(* IEC 61131-3 sources: AXOpen/src/components.festo.drives/ctrl/src/PROFIdrive, 6 files *)

(* ---- AxoPROFIdriveParametrization.st ---- *)
USING AXOpen.Core;
USING Siemens.Simatic.DistributedIO;

NAMESPACE AXOpen.Components.Festo.Drives
    {S7.extern=ReadWrite}
    CLASS AxoPROFIdriveParametrization
        VAR PUBLIC
            {#ix-attr:[Container(Layout.Wrap)]}
            {#ix-attr:[Group(GroupLayout.GroupBox)]}
            {#ix-set:AttributeName = "<#Inputs#>"}
            Inputs				:	AxoPROFIdriveParametrizationIn;
            {#ix-attr:[Container(Layout.Wrap)]}
            {#ix-attr:[Group(GroupLayout.GroupBox)]}
            {#ix-set:AttributeName = "<#Outputs#>"}
            {#ix-attr:[ReadOnly()]}
            Outputs				:	AxoPROFIdriveParametrizationOut;
        END_VAR
    END_CLASS
END_NAMESPACE

(* ---- AxoPROFIdriveParametrizationIn.st ---- *)
USING AXOpen.Core;
USING Siemens.Simatic.DistributedIO;

NAMESPACE AXOpen.Components.Festo.Drives
    {S7.extern=ReadWrite}
    CLASS AxoPROFIdriveParametrizationIn
        VAR PUBLIC
            {#ix-attr:[Container(Layout.Stack)]}
            {#ix-set:AttributeName = "<#Enable#>"}
            Enable          :   BOOL;
            {#ix-set:AttributeName = "<#ReadWrite#>"}
            ReadWrite       :   BOOL;
            {#ix-set:AttributeName = "<#ParameterNo#>"}
            ParameterNo     :   INT;
            {#ix-set:AttributeName = "<#Subindex#>"}
            Subindex        :   INT;
            {#ix-set:AttributeName = "<#AxisNo#>"}
            AxisNo	        :   BYTE := BYTE#1;
            {#ix-set:AttributeName = "<#HardwareId#>"}
            HardwareId	    :   UINT;
            {#ix-set:AttributeName = "<#ValueWriteREAL#>"}
            ValueWriteREAL  :   REAL;
            {#ix-set:AttributeName = "<#ValueWriteLINT#>"}
            ValueWriteLINT  :   LINT;
            {#ix-set:AttributeName = "<#ValueWriteBOOL#>"}
            ValueWriteBOOL  :   BOOL;
        END_VAR
    END_CLASS
END_NAMESPACE

(* ---- AxoPROFIdriveParametrizationOut.st ---- *)
USING AXOpen.Core;
USING Siemens.Simatic.DistributedIO;

NAMESPACE AXOpen.Components.Festo.Drives
    {S7.extern=ReadWrite}
    CLASS AxoPROFIdriveParametrizationOut
        VAR PUBLIC
            {#ix-attr:[Container(Layout.Stack)]}
            {#ix-set:AttributeName = "<#ValueReadREAL#>"}
            ValueReadREAL  :   REAL;
            {#ix-set:AttributeName = "<#ValueReadLINT#>"}
            ValueReadLINT  :   LINT;
            {#ix-set:AttributeName = "<#ValueReadBOOL#>"}
            ValueReadBOOL  :   BOOL;
            {#ix-set:AttributeName = "<#Busy#>"}
            Busy	:   BOOL;
            {#ix-set:AttributeName = "<#Done#>"}
            Done	:   BOOL;
            {#ix-set:AttributeName = "<#Error#>"}
            Error	:   BOOL;
            {#ix-set:AttributeName = "<#ErrorId#>"}
            ErrorId :	DWORD;
        END_VAR

    END_CLASS
END_NAMESPACE

(* ---- AxoReadWritePROFIdriveParameter.st ---- *)
USING AXOpen.Core;
USING Siemens.Simatic.S71500.DistributedIO;

NAMESPACE AXOpen.Components.Festo.Drives
    {S7.extern=ReadWrite}
    CLASS AxoReadWritePROFIdriveParameter EXTENDS AXOpen.Core.AxoObject
        VAR PUBLIC
            {#ix-attr:[Container(Layout.Wrap)]}
            {#ix-attr:[Group(GroupLayout.GroupBox)]}
            {#ix-set:AttributeName = "<#Inputs#>"}
            Inputs				:	AxoPROFIdriveParametrizationIn;
            {#ix-attr:[Container(Layout.Wrap)]}
            {#ix-attr:[Group(GroupLayout.GroupBox)]}
            {#ix-set:AttributeName = "<#Outputs#>"}
            {#ix-attr:[ReadOnly()]}
            Outputs				:	AxoPROFIdriveParametrizationOut;
        END_VAR

        VAR PRIVATE
            Enable_PV   :   BOOL;

            Busy_	:   BOOL;
            Done_	:   BOOL;
            Error_	:   BOOL;
            ErrorId_:	DWORD;
            StartTimer : BOOL;
            StartRW : BOOL;

            AxoOnDelatTimer :  AXOpen.Timers.OnDelayTimer;

            RW_Data         :   ARRAY[0..9] OF BYTE;
            WR_Data         :   ARRAY[0..19] OF BYTE;
            RD_Data         :   ARRAY[0..13] OF BYTE;
            RW_Status        :	DWORD;
            WR_Status        :	DWORD;
            RD_Status        :	DWORD;

            ReadRecord_     :   ReadRecord;
            WriteRecord_    :   WriteRecord;
            ErrorCounter    :	UINT;

            LengthRead      :	UINT;
            State           :   INT;
            ReqRef          :   BYTE;
            wordhlp         :   WORD;

            _lenght     :   UINT;
            tmpWord     :   WORD;
            tmpSINT     :   SINT;
            tmpINT      :   INT;
            tmpDINT     :   DINT;
            tmpDWORD    :   DWORD;
            tmpLINT     :   LINT;
        END_VAR

        VAR CONSTANT PRIVATE
            LenHeader	    :   UINT    :=	UINT#4;
            LenRequest	    :   UINT    :=  UINT#6;
            LenWrite	    :   UINT    :=  UINT#16;
            LenRead	        :   UINT    :=  UINT#10;
            PD_Error	    :   DWORD	:=  DWORD#16#4000_0000;
            MaxRetryCounter	:   UINT    :=	UINT#150;

        END_VAR

        METHOD PUBLIC OVERRIDE Run
            VAR_INPUT
                inParent : IAxoObject;
            END_VAR
            VAR
                i : INT;
            END_VAR

            SUPER.Run(inParent);

            //**********************************************
            // THIS.Execute();
            //*****************Execute inline***************
                //Check the Inputs
                IF Inputs.HardwareId = WORD#0 THEN
                    Error_ := TRUE;
                    ErrorId_ := DWORD#16#00001010;    //Inputs.HardwareId = 0
                    RETURN;
                END_IF;

                //Timer
                AxoOnDelatTimer.OnDelay(THIS, StartTimer,T#100MS);

                IF AxoOnDelatTimer.output THEN
                    StartRW := TRUE;
                    StartTimer := FALSE;
                END_IF;

                IF State = 0 THEN //Wait for start trigger
                    IF Inputs.Enable AND NOT Enable_PV THEN
                        StartRW := TRUE;
                        State := 10;
                        Outputs.Busy := TRUE;
                    END_IF;
                END_IF;

                IF State = 10 THEN
                    (* ------------------ HEADER --------------------*)
                    //Request reference starts with 1 and will count up
                    RW_Data[0] := ReqRef;
                    // Requst ID = 1 (Request Parameter)
                    RW_Data[1] := BYTE#1;
                    //Fill the Axis number
                    RW_Data[2] := Inputs.AxisNo;
                    // Single parameter access
                    RW_Data[3] := BYTE#1;
                    (* ------------------ Parameter address ------------*)
                    //Attribute
                    RW_Data[4]:= BYTE#16#10;
                    //ElemNo.
                    RW_Data[5] := BYTE#1;
                    // Assign PNU
                    RW_Data[6] := Inputs.ParameterNo.%B1;
                    RW_Data[7] := Inputs.ParameterNo.%B0;
                    // Assign Subindex
                    RW_Data[8] := Inputs.Subindex.%B1;
                    RW_Data[9] := Inputs.Subindex.%B0;

                    // Lenght of the telegramm to be send
                    _lenght := LenHeader + LenRequest;

                    WriteRecord_(request    :=  StartRW,
                                id          :=  Inputs.HardwareId,
                                index       :=  16#b02e,
                                length      :=  _lenght,
                                record      :=  RW_Data,
                                status      =>  WR_Status);

                    IF WriteRecord_.DONE THEN
                        ErrorCounter := UINT#0;
                        //delete old response values
                        FOR i := 0 TO 13 DO
                            RD_Data[i] := BYTE#0;
                        END_FOR;

                        IF NOT Inputs.ReadWrite THEN
                            //Read parameter
                            State := 20;
                        ELSE
                            //Write parameter
                            State := 50;
                        END_IF;
                    ELSIF WriteRecord_.ERROR THEN
                        tmpWord := TO_WORD(TO_DINT(WR_Status)/256);
                        wordhlp := tmpWord;
                        //try it again
                        IF ((tmpWord = WORD#16#80A7) OR (tmpWord = WORD#16#80B5) OR (tmpWord = WORD#16#80C0) OR (tmpWord = WORD#16#80C1) OR (tmpWord = WORD#16#80C2)
                            OR (tmpWord = WORD#16#80C3) OR (tmpWord = WORD#16#80C4)) AND (ErrorCounter < MaxRetryCounter) THEN
                            ErrorCounter := ErrorCounter + UINT#1;
                            StartRW := FALSE;
                            StartTimer := TRUE;
                        ELSE
                            State := 70;
                        END_IF;

                    END_IF;
                END_IF;

                IF State = 20 THEN  //Read Parameter
                    // Lenght of the telegramm for reading
                    _lenght := LenHeader + LenRead;

                    ReadRecord_(request     :=  StartRW,
                                id          :=  Inputs.HardwareId,
                                index       :=  16#b02e,
                                maxLength   :=  _lenght,
                                record      :=  RD_Data,
                                status      =>  RD_Status,
                                length      =>  LengthRead);

                    IF ReadRecord_.VALID AND NOT ReadRecord_.BUSY THEN
                        ErrorCounter := UINT#0;
                        State := 30;
                    ELSIF ReadRecord_.ERROR THEN
                        tmpWord := TO_WORD(TO_DINT(RD_Status) / 256);
                        wordhlp := tmpWord;
                        //try it again
                        IF ((tmpWord = WORD#16#80A7) OR (tmpWord = WORD#16#80B5) OR (tmpWord = WORD#16#80C0) OR (tmpWord = WORD#16#80C1) OR (tmpWord = WORD#16#80C2)
                            OR (tmpWord = WORD#16#80C3) OR (tmpWord = WORD#16#80C4)) AND (ErrorCounter < MaxRetryCounter) THEN
                            ErrorCounter := ErrorCounter + UINT#1;
                            StartRW := FALSE;
                            StartTimer := TRUE;
                        ELSE
                            State := 80;
                        END_IF;
                    END_IF;
                END_IF;

                IF State = 30 THEN //Reading finished successfull

                    CASE TO_INT(RD_Data[4]) OF //Format
                        0:  //reserved
                            Outputs.ValueReadREAL := REAL#0.0;
                            Outputs.ValueReadLINT := LINT#0;
                            Outputs.ValueReadBOOL := FALSE;

                            Outputs.ErrorId := DWORD#16#1001;    //reserved DataType
                            // #Error
                            State := 200;

                        1:  // BOOLEAN
                            //copy the value to the output
                            Outputs.ValueReadREAL := 0;
                            Outputs.ValueReadLINT := 0;
                            Outputs.ValueReadBOOL := TO_BOOL(RD_Data[6]);

                            // no error
                            State := 100;

                        2:  //SINT8
                            tmpSINT := TO_SINT(RD_Data[6]);
                            //copy the value to the output
                            Outputs.ValueReadREAL := 0;
                            Outputs.ValueReadLINT := (TO_LINT(tmpSINT));
                            Outputs.ValueReadBOOL := FALSE;

                            // no error
                            State := 100;

                        3:  //SINT16
                            tmpINT.%B0 := RD_Data[7];
                            tmpINT.%B1 := RD_Data[6];

                            //copy the value to the output
                            Outputs.ValueReadREAL := 0;
                            Outputs.ValueReadLINT := TO_LINT(tmpINT);
                            Outputs.ValueReadBOOL := FALSE;

                            // no #Error
                            State := 100;

                        4:  //SINT32
                            tmpDINT.%B0 := RD_Data[9];
                            tmpDINT.%B1 := RD_Data[8];
                            tmpDINT.%B2 := RD_Data[7];
                            tmpDINT.%B3 := RD_Data[6];

                            //copy the value to the output
                            Outputs.ValueReadREAL := 0;
                            Outputs.ValueReadLINT := TO_LINT(tmpDINT);
                            Outputs.ValueReadBOOL := FALSE;

                            // no #Error
                            State := 100;

                        5, 65: //USINT8(5) or BYTE(65)
                            //copy the value to the output
                            Outputs.ValueReadREAL := 0;
                            Outputs.ValueReadLINT := (TO_LINT(RD_Data[6]));
                            Outputs.ValueReadBOOL := FALSE;

                            // no error
                            State := 100;

                        6, 66: //UINT16(6) or WORD(66)
                            tmpWord.%B0 := RD_Data[7];
                            tmpWord.%B1 := RD_Data[6];

                            //copy the value to the output
                            Outputs.ValueReadREAL := 0;
                            Outputs.ValueReadLINT := TO_LINT(tmpWord);
                            Outputs.ValueReadBOOL := FALSE;

                            // no #Error
                            State := 100;

                        7, 67: //UDINT32(7) or DWORD(67)
                            tmpDWord.%B0 := RD_Data[9];
                            tmpDWord.%B1 := RD_Data[8];
                            tmpDWord.%B2 := RD_Data[7];
                            tmpDWord.%B3 := RD_Data[6];

                            //copy the value to the output
                            Outputs.ValueReadREAL := 0;
                            Outputs.ValueReadLINT := TO_LINT(tmpDWord);
                            Outputs.ValueReadBOOL := FALSE;

                            // no #Error
                            State := 100;

                        8:  //FLOAT32
                            tmpDWord.%B0 := RD_Data[9];
                            tmpDWord.%B1 := RD_Data[8];
                            tmpDWord.%B2 := RD_Data[7];
                            tmpDWord.%B3 := RD_Data[6];

                            //copy the value to the output
                            Outputs.ValueReadREAL := TO_REAL(tmpDWord);
                            Outputs.ValueReadLINT := 0;
                            Outputs.ValueReadBOOL := FALSE;

                            // no #Error
                            State := 100;

                        10:  //OctetString
                            tmpINT.%B0 := RD_Data[6];
                            tmpINT.%B1 := RD_Data[7];

                            //copy the value to the output
                            Outputs.ValueReadREAL := 0;
                            Outputs.ValueReadLINT := TO_LINT(tmpINT);
                            Outputs.ValueReadBOOL := FALSE;

                            // no #Error
                            State := 100;

                        55, 56:  //LINT, ULINT
                            tmpLINT.%B0 :=RD_Data[13];
                            tmpLINT.%B1 :=RD_Data[12];
                            tmpLINT.%B2 :=RD_Data[11];
                            tmpLINT.%B3 :=RD_Data[10];
                            tmpLINT.%B4 :=RD_Data[9];
                            tmpLINT.%B5 :=RD_Data[8];
                            tmpLINT.%B6 :=RD_Data[7];
                            tmpLINT.%B7 :=RD_Data[6];

                            //copy the value to the output
                            Outputs.ValueReadREAL := 0;
                            Outputs.ValueReadLINT := tmpLINT;
                            Outputs.ValueReadBOOL := FALSE;

                            // no #Error
                            State := 100;

                        68:  //Error
                            tmpDWord.%B0 := RD_Data[7];
                            tmpDWord.%B1 := RD_Data[6];
                            Outputs.ErrorId := tmpDWord OR PD_Error;

                            //copy the value to the output
                            Outputs.ValueReadREAL := 0;
                            Outputs.ValueReadLINT := 0;
                            Outputs.ValueReadBOOL := FALSE;

                            // #Error
                            State := 200;

                        ELSE
                            Outputs.ValueReadREAL := 0;
                            Outputs.ValueReadLINT := 0;
                            Outputs.ValueReadBOOL := FALSE;

                            Outputs.ErrorId := DWORD#16#1000;    //unknown DataType
                            // #Error
                            State := 200;
                    END_CASE;
                END_IF;

                IF State = 50 THEN //Write Parameter (First Read dataset then write dataset)
                    // Lenght of the telegramm for reading
                    _lenght := LenHeader + LenRead;

                    ReadRecord_(request     :=  StartRW,
                                id          :=  Inputs.HardwareId,
                                index       :=  16#b02e,
                                maxLength   :=  _lenght,
                                record      :=  RD_Data,
                                status      =>  RD_Status,
                                length      =>  LengthRead);

                    IF ReadRecord_.VALID AND NOT ReadRecord_.BUSY THEN
                        ErrorCounter := UINT#0;
                        State := 55;
                    ELSIF ReadRecord_.ERROR THEN
                        tmpWord := TO_WORD(TO_DINT(RD_Status)/256);
                        wordhlp := tmpWord;
                        //try it again
                        IF ((tmpWord = WORD#16#80A7) OR (tmpWord = WORD#16#80B5) OR (tmpWord = WORD#16#80C0) OR (tmpWord = WORD#16#80C1) OR (tmpWord = WORD#16#80C2)
                            OR (tmpWord = WORD#16#80C3) OR (tmpWord = WORD#16#80C4)) AND (ErrorCounter < MaxRetryCounter) THEN
                            ErrorCounter := ErrorCounter + UINT#1;
                            StartRW := false;
                            StartTimer := TRUE;
                        ELSE
                            State := 80;
                        END_IF;
                    END_IF;
                END_IF;

                IF State = 55 THEN //Reading finished
                    CASE TO_INT(RD_Data[4]) OF // Format
                        0:  //reserved
                            Outputs.ValueReadREAL := 0;
                            Outputs.ValueReadLINT := 0;
                            Outputs.ValueReadBOOL := FALSE;

                            Outputs.ErrorId := DWORD#16#1001;    //reserved DataType
                            // #Error
                            State := 200;

                        1, 2, 3, 4, 5, 6, 7, 8, 55, 56, 65, 66, 67:
                            State := 60;

                        68:  //Error
                            tmpDWord.%B0 := RD_Data[7];
                            tmpDWord.%B1 := RD_Data[6];
                            Outputs.ErrorId := tmpDWord OR PD_Error;

                            //copy the value to the output
                            Outputs.ValueReadREAL := 0;
                            Outputs.ValueReadLINT := 0;
                            Outputs.ValueReadBOOL := FALSE;

                            // #Error
                            State := 200;

                        ELSE
                            Outputs.ValueReadREAL := 0;
                            Outputs.ValueReadLINT := 0;
                            Outputs.ValueReadBOOL := FALSE;

                            Outputs.ErrorId := DWORD#16#1000;    //unknown DataType
                            // #Error
                            State := 200;
                    END_CASE;
                END_IF;

                IF State = 60 THEN //reading Done from Write request
                    (* ------------------ HEADER --------------------*)
                    //Request reference starts with 1 and will count up
                    WR_Data[0] := TO_BYTE(TO_INT(ReqRef) + 1);
                    // Requst ID = 2 (Change Parameter)
                    WR_Data[1] := BYTE#2;
                    //Fill the Axis number
                    WR_Data[2] := Inputs.AxisNo;
                    // Single parameter access
                    WR_Data[3] := BYTE#1;
                    (* ------------------ DATA --------------------*)
                    // Attribute
                    WR_Data[4] := BYTE#16#10;
                    // Single Access
                    WR_Data[5] := BYTE#1;
                    // PNU
                    WR_Data[6] := Inputs.ParameterNo.%B1;
                    WR_Data[7] := Inputs.ParameterNo.%B0;
                    // Subindex
                    WR_Data[8] := Inputs.Subindex.%B1;
                    WR_Data[9] := Inputs.Subindex.%B0;
                    //Format
                    WR_Data[10] := RD_Data[4];
                    //No. Values
                    WR_Data[11] := BYTE#1;
                    //erase send buffer
                    FOR i := 12 TO 19 DO
                        WR_Data[i] := BYTE#0;
                    END_FOR;

                    CASE TO_INT(RD_Data[4]) OF //Format
                        0:  //reserved
                            Outputs.ValueReadREAL := 0;
                            Outputs.ValueReadLINT := 0;
                            Outputs.ValueReadBOOL := FALSE;

                            Outputs.ErrorId := DWORD#16#1001;    //reserved DataType
                            // #Error
                            State := 200;

                        1:  //BOOL
                            WR_Data[12] := TO_BYTE(Inputs.ValueWriteBOOL);

                        2, 5, 65:  //SINT8, USINT8, BYTE
                            WR_Data[12] := TO_BYTE(Inputs.ValueWriteLINT);

                        3, 6, 66:  //SINT16, UINT16, WORD
                            WR_Data[12] := Inputs.ValueWriteLINT.%B1;
                            WR_Data[13] := Inputs.ValueWriteLINT.%B0;

                        4, 7, 67: //SINT32, UDINT32, DWORD
                            WR_Data[12] := Inputs.ValueWriteLINT.%B3;
                            WR_Data[13] := Inputs.ValueWriteLINT.%B2;
                            WR_Data[14] := Inputs.ValueWriteLINT.%B1;
                            WR_Data[15] := Inputs.ValueWriteLINT.%B0;

                        8:  //FLOAT32
                            tmpDWORD    :=  TO_DWORD(Inputs.ValueWriteREAL);
                            WR_Data[12] := tmpDWORD.%B3;
                            WR_Data[13] := tmpDWORD.%B2;
                            WR_Data[14] := tmpDWORD.%B1;
                            WR_Data[15] := tmpDWORD.%B0;

                        55, 56:  //SINT64
                            WR_Data[12] := Inputs.ValueWriteLINT.%B7;
                            WR_Data[13] := Inputs.ValueWriteLINT.%B6;
                            WR_Data[14] := Inputs.ValueWriteLINT.%B5;
                            WR_Data[15] := Inputs.ValueWriteLINT.%B4;
                            WR_Data[16] := Inputs.ValueWriteLINT.%B3;
                            WR_Data[17] := Inputs.ValueWriteLINT.%B2;
                            WR_Data[18] := Inputs.ValueWriteLINT.%B1;
                            WR_Data[19] := Inputs.ValueWriteLINT.%B0;

                    END_CASE;

                    //goto the next step
                    State := 61;
                END_IF;

                IF State = 61 THEN //send the write Request
                    // Lenght of the telegramm to be send
                    _lenght := LenHeader + LenWrite;

                    WriteRecord_(request    :=  StartRW,
                                id          :=  Inputs.HardwareId,
                                index       :=  16#b02e,
                                length      :=  _lenght,
                                record      :=  WR_Data,
                                status      =>  RW_Status);

                    IF WriteRecord_.DONE THEN
                        State := 62;
                    ELSIF WriteRecord_.ERROR THEN
                        tmpWord := TO_WORD(TO_DINT(RW_Status)/256);
                        wordhlp := tmpWord;
                        //try it again
                        IF ((tmpWord = WORD#16#80A7) OR (tmpWord = WORD#16#80B5) OR (tmpWord = WORD#16#80C0) OR (tmpWord = WORD#16#80C1) OR (tmpWord = WORD#16#80C2)
                            OR (tmpWord = WORD#16#80C3) OR (tmpWord = WORD#16#80C4)) AND (ErrorCounter < MaxRetryCounter) THEN
                            ErrorCounter := ErrorCounter + UINT#1;
                            StartRW := FALSE;
                            StartTimer := TRUE;
                        ELSE
                            State := 90;
                        END_IF;
                    END_IF;
                END_IF;

                IF State = 62 THEN //Read the answer of the write request

                    //delete old response values
                    FOR i := 0 TO 13 DO
                        RD_Data[i] := BYTE#0;
                    END_FOR;

                    // Lenght of the telegramm for reading
                    _lenght := LenHeader + LenRead;

                    ReadRecord_(request     :=  StartRW,
                                id          :=  Inputs.HardwareId,
                                index       :=  16#b02e,
                                maxLength   :=  _lenght,
                                record      :=  RD_Data,
                                status      =>  RD_Status,
                                length      =>  LengthRead);

                    IF ReadRecord_.VALID AND NOT ReadRecord_.BUSY THEN
                        ErrorCounter := UINT#0;
                        State := 63;
                    ELSIF ReadRecord_.ERROR THEN
                        tmpWord := TO_WORD(TO_DINT(RD_Status)/256);
                        wordhlp := tmpWord;
                        //try it again
                        IF ((tmpWord = WORD#16#80A7) OR (tmpWord = WORD#16#80B5) OR (tmpWord = WORD#16#80C0) OR (tmpWord = WORD#16#80C1) OR (tmpWord = WORD#16#80C2)
                            OR (tmpWord = WORD#16#80C3) OR (tmpWord = WORD#16#80C4)) AND (ErrorCounter < MaxRetryCounter) THEN
                            ErrorCounter := ErrorCounter + UINT#1;
                            StartRW := FALSE;
                            StartTimer := TRUE;
                        ELSE
                            State := 80;
                        END_IF;
                    END_IF;
                END_IF;

                IF State = 63 THEN //Reading finished

                    CASE TO_INT(RD_Data[1]) OF //ReqId

                        2:  //positive resonse
                            State := 150;

                        128..130:  //negative response
                            IF RD_Data[4] = BYTE#68 THEN //Format
                                tmpDWord.%B0 := RD_Data[7];
                                tmpDWord.%B1 := RD_Data[6];
                                Outputs.ErrorId := tmpDWord OR PD_Error;

                                // #Error
                                State := 200;
                            ELSE
                                Outputs.ErrorId := DWORD#16#1003; //negative response without error code
                                State := 300;
                            END_IF;
                        ELSE  //undefined response ID
                            Outputs.ErrorId := DWORD#16#1002;
                            State := 300;
                    END_CASE;
                END_IF;

                IF State = 70 THEN // Error while ReadWrite Access
                    Outputs.Done := TRUE;
                    Outputs.Busy := FALSE;
                    Outputs.Error := TRUE;
                    Outputs.ErrorId := WR_Status;
                END_IF;

                IF State = 80 THEN //Error Reading Access
                    Outputs.Done := TRUE;
                    Outputs.Busy := FALSE;
                    Outputs.Error := TRUE;
                    Outputs.ErrorId := RD_Status;
                END_IF;

                IF State = 90 THEN // Error while Write Access
                    Outputs.Done := TRUE;
                    Outputs.Busy := FALSE;
                    Outputs.Error := TRUE;
                    Outputs.ErrorId := RW_Status;
                END_IF;

                IF State = 100 THEN // read successfully
                    Outputs.Done := TRUE;
                    Outputs.Busy := FALSE;
                    Outputs.Error := FALSE;
                END_IF;

                IF State = 150 THEN // write successfully
                    Outputs.Done := TRUE;
                    Outputs.Busy := FALSE;
                    Outputs.Error := FALSE;
                END_IF;

                IF State = 200 THEN //Error while reading
                    Outputs.Done := TRUE;
                    Outputs.Busy := FALSE;
                    Outputs.Error := TRUE;

                    IF State = 300 THEN //Error while writing
                        Outputs.Done := TRUE;
                        Outputs.Busy := FALSE;
                        Outputs.Error := TRUE;
                    END_IF;
                END_IF;

                IF NOT Inputs.Enable THEN
                    State := 0;
                    ReqRef := BYTE#1;
                    Outputs.Done := FALSE;
                    Outputs.Busy := FALSE;
                    Outputs.Error := FALSE;
                    Outputs.ErrorId := DWORD#16#00000000;
                    Outputs.ValueReadBOOL := FALSE;
                    Outputs.ValueReadLINT := 0;
                    Outputs.ValueReadREAL := 0;
                    RD_Status := DWORD#0;
                    ErrorCounter := UINT#0;
                END_IF;

                Enable_PV := Inputs.Enable;

        END_METHOD

        // METHOD PUBLIC Execute

        //     VAR
        //         _lenght     :   UINT;
        //         i           :   INT;
        //         tmpWord     :   WORD;
        //         tmpSINT     :   SINT;
        //         tmpINT      :   INT;
        //         tmpDINT     :   DINT;
        //         tmpDWORD    :   DWORD;
        //         tmpLINT     :   LINT;
        //     END_VAR

        //         //Check the Inputs
        //         IF Inputs.HardwareId = WORD#0 THEN
        //             Error_ := TRUE;
        //             ErrorId_ := DWORD#16#00001010;    //Inputs.HardwareId = 0
        //             RETURN;
        //         END_IF;

        //         //Timer
        //         AxoOnDelatTimer.OnDelay(THIS, StartTimer,T#100MS);

        //         IF AxoOnDelatTimer.output THEN
        //             StartRW := TRUE;
        //             StartTimer := FALSE;
        //         END_IF;

        //         IF State = 0 THEN //Wait for start trigger
        //             IF Inputs.Enable AND NOT Enable_PV THEN
        //                 StartRW := TRUE;
        //                 State := 10;
        //                 Outputs.Busy := TRUE;
        //             END_IF;
        //         END_IF;

        //         IF State = 10 THEN
        //             (* ------------------ HEADER --------------------*)
        //             //Request reference starts with 1 and will count up
        //             RW_Data[0] := ReqRef;
        //             // Requst ID = 1 (Request Parameter)
        //             RW_Data[1] := BYTE#1;
        //             //Fill the Axis number
        //             RW_Data[2] := Inputs.AxisNo;
        //             // Single parameter access
        //             RW_Data[3] := BYTE#1;
        //             (* ------------------ Parameter address ------------*)
        //             //Attribute
        //             RW_Data[4]:= BYTE#16#10;
        //             //ElemNo.
        //             RW_Data[5] := BYTE#1;
        //             // Assign PNU
        //             RW_Data[6] := Inputs.ParameterNo.%B1;
        //             RW_Data[7] := Inputs.ParameterNo.%B0;
        //             // Assign Subindex
        //             RW_Data[8] := Inputs.Subindex.%B1;
        //             RW_Data[9] := Inputs.Subindex.%B0;

        //             // Lenght of the telegramm to be send
        //             _lenght := LenHeader + LenRequest;

        //             WriteRecord_(request    :=  StartRW,
        //                         id          :=  Inputs.HardwareId,
        //                         index       :=  16#b02e,
        //                         length      :=  _lenght,
        //                         record      :=  RW_Data,
        //                         status      =>  WR_Status);

        //             IF WriteRecord_.DONE THEN
        //                 ErrorCounter := UINT#0;
        //                 //delete old response values
        //                 FOR i := 0 TO 13 DO
        //                     RD_Data[i] := BYTE#0;
        //                 END_FOR;

        //                 IF NOT Inputs.ReadWrite THEN
        //                     //Read parameter
        //                     State := 20;
        //                 ELSE
        //                     //Write parameter
        //                     State := 50;
        //                 END_IF;
        //             ELSIF WriteRecord_.ERROR THEN
        //                 tmpWord := TO_WORD(TO_DINT(WR_Status)/256);
        //                 wordhlp := tmpWord;
        //                 //try it again
        //                 IF ((tmpWord = WORD#16#80A7) OR (tmpWord = WORD#16#80B5) OR (tmpWord = WORD#16#80C0) OR (tmpWord = WORD#16#80C1) OR (tmpWord = WORD#16#80C2)
        //                     OR (tmpWord = WORD#16#80C3) OR (tmpWord = WORD#16#80C4)) AND (ErrorCounter < MaxRetryCounter) THEN
        //                     ErrorCounter := ErrorCounter + UINT#1;
        //                     StartRW := FALSE;
        //                     StartTimer := TRUE;
        //                 ELSE
        //                     State := 70;
        //                 END_IF;

        //             END_IF;
        //         END_IF;

        //         IF State = 20 THEN  //Read Parameter
        //             // Lenght of the telegramm for reading
        //             _lenght := LenHeader + LenRead;

        //             ReadRecord_(request     :=  StartRW,
        //                         id          :=  Inputs.HardwareId,
        //                         index       :=  16#b02e,
        //                         maxLength   :=  _lenght,
        //                         record      :=  RD_Data,
        //                         status      =>  RD_Status,
        //                         length      =>  LengthRead);

        //             IF ReadRecord_.VALID AND NOT ReadRecord_.BUSY THEN
        //                 ErrorCounter := UINT#0;
        //                 State := 30;
        //             ELSIF ReadRecord_.ERROR THEN
        //                 tmpWord := TO_WORD(TO_DINT(RD_Status) / 256);
        //                 wordhlp := tmpWord;
        //                 //try it again
        //                 IF ((tmpWord = WORD#16#80A7) OR (tmpWord = WORD#16#80B5) OR (tmpWord = WORD#16#80C0) OR (tmpWord = WORD#16#80C1) OR (tmpWord = WORD#16#80C2)
        //                     OR (tmpWord = WORD#16#80C3) OR (tmpWord = WORD#16#80C4)) AND (ErrorCounter < MaxRetryCounter) THEN
        //                     ErrorCounter := ErrorCounter + UINT#1;
        //                     StartRW := FALSE;
        //                     StartTimer := TRUE;
        //                 ELSE
        //                     State := 80;
        //                 END_IF;
        //             END_IF;
        //         END_IF;

        //         IF State = 30 THEN //Reading finished successfull

        //             CASE TO_INT(RD_Data[4]) OF //Format
        //                 0:  //reserved
        //                     Outputs.ValueReadREAL := REAL#0.0;
        //                     Outputs.ValueReadLINT := LINT#0;
        //                     Outputs.ValueReadBOOL := FALSE;

        //                     Outputs.ErrorId := DWORD#16#1001;    //reserved DataType
        //                     // #Error
        //                     State := 200;

        //                 1:  // BOOLEAN
        //                     //copy the value to the output
        //                     Outputs.ValueReadREAL := 0;
        //                     Outputs.ValueReadLINT := 0;
        //                     Outputs.ValueReadBOOL := TO_BOOL(RD_Data[6]);

        //                     // no error
        //                     State := 100;

        //                 2:  //SINT8
        //                     tmpSINT := TO_SINT(RD_Data[6]);
        //                     //copy the value to the output
        //                     Outputs.ValueReadREAL := 0;
        //                     Outputs.ValueReadLINT := (TO_LINT(tmpSINT));
        //                     Outputs.ValueReadBOOL := FALSE;

        //                     // no error
        //                     State := 100;

        //                 3:  //SINT16
        //                     tmpINT.%B0 := RD_Data[7];
        //                     tmpINT.%B1 := RD_Data[6];

        //                     //copy the value to the output
        //                     Outputs.ValueReadREAL := 0;
        //                     Outputs.ValueReadLINT := TO_LINT(tmpINT);
        //                     Outputs.ValueReadBOOL := FALSE;

        //                     // no #Error
        //                     State := 100;

        //                 4:  //SINT32
        //                     tmpDINT.%B0 := RD_Data[9];
        //                     tmpDINT.%B1 := RD_Data[8];
        //                     tmpDINT.%B2 := RD_Data[7];
        //                     tmpDINT.%B3 := RD_Data[6];

        //                     //copy the value to the output
        //                     Outputs.ValueReadREAL := 0;
        //                     Outputs.ValueReadLINT := TO_LINT(tmpDINT);
        //                     Outputs.ValueReadBOOL := FALSE;

        //                     // no #Error
        //                     State := 100;

        //                 5, 65: //USINT8(5) or BYTE(65)
        //                     //copy the value to the output
        //                     Outputs.ValueReadREAL := 0;
        //                     Outputs.ValueReadLINT := (TO_LINT(RD_Data[6]));
        //                     Outputs.ValueReadBOOL := FALSE;

        //                     // no error
        //                     State := 100;

        //                 6, 66: //UINT16(6) or WORD(66)
        //                     tmpWord.%B0 := RD_Data[7];
        //                     tmpWord.%B1 := RD_Data[6];

        //                     //copy the value to the output
        //                     Outputs.ValueReadREAL := 0;
        //                     Outputs.ValueReadLINT := TO_LINT(tmpWord);
        //                     Outputs.ValueReadBOOL := FALSE;

        //                     // no #Error
        //                     State := 100;

        //                 7, 67: //UDINT32(7) or DWORD(67)
        //                     tmpDWord.%B0 := RD_Data[9];
        //                     tmpDWord.%B1 := RD_Data[8];
        //                     tmpDWord.%B2 := RD_Data[7];
        //                     tmpDWord.%B3 := RD_Data[6];

        //                     //copy the value to the output
        //                     Outputs.ValueReadREAL := 0;
        //                     Outputs.ValueReadLINT := TO_LINT(tmpDWord);
        //                     Outputs.ValueReadBOOL := FALSE;

        //                     // no #Error
        //                     State := 100;

        //                 8:  //FLOAT32
        //                     tmpDWord.%B0 := RD_Data[9];
        //                     tmpDWord.%B1 := RD_Data[8];
        //                     tmpDWord.%B2 := RD_Data[7];
        //                     tmpDWord.%B3 := RD_Data[6];

        //                     //copy the value to the output
        //                     Outputs.ValueReadREAL := TO_REAL(tmpDWord);
        //                     Outputs.ValueReadLINT := 0;
        //                     Outputs.ValueReadBOOL := FALSE;

        //                     // no #Error
        //                     State := 100;

        //                 10:  //OctetString
        //                     tmpINT.%B0 := RD_Data[6];
        //                     tmpINT.%B1 := RD_Data[7];

        //                     //copy the value to the output
        //                     Outputs.ValueReadREAL := 0;
        //                     Outputs.ValueReadLINT := TO_LINT(tmpINT);
        //                     Outputs.ValueReadBOOL := FALSE;

        //                     // no #Error
        //                     State := 100;

        //                 55, 56:  //LINT, ULINT
        //                     tmpLINT.%B0 :=RD_Data[13];
        //                     tmpLINT.%B1 :=RD_Data[12];
        //                     tmpLINT.%B2 :=RD_Data[11];
        //                     tmpLINT.%B3 :=RD_Data[10];
        //                     tmpLINT.%B4 :=RD_Data[9];
        //                     tmpLINT.%B5 :=RD_Data[8];
        //                     tmpLINT.%B6 :=RD_Data[7];
        //                     tmpLINT.%B7 :=RD_Data[6];

        //                     //copy the value to the output
        //                     Outputs.ValueReadREAL := 0;
        //                     Outputs.ValueReadLINT := tmpLINT;
        //                     Outputs.ValueReadBOOL := FALSE;

        //                     // no #Error
        //                     State := 100;

        //                 68:  //Error
        //                     tmpDWord.%B0 := RD_Data[7];
        //                     tmpDWord.%B1 := RD_Data[6];
        //                     Outputs.ErrorId := tmpDWord OR PD_Error;

        //                     //copy the value to the output
        //                     Outputs.ValueReadREAL := 0;
        //                     Outputs.ValueReadLINT := 0;
        //                     Outputs.ValueReadBOOL := FALSE;

        //                     // #Error
        //                     State := 200;

        //                 ELSE
        //                     Outputs.ValueReadREAL := 0;
        //                     Outputs.ValueReadLINT := 0;
        //                     Outputs.ValueReadBOOL := FALSE;

        //                     Outputs.ErrorId := DWORD#16#1000;    //unknown DataType
        //                     // #Error
        //                     State := 200;
        //             END_CASE;
        //         END_IF;

        //         IF State = 50 THEN //Write Parameter (First Read dataset then write dataset)
        //             // Lenght of the telegramm for reading
        //             _lenght := LenHeader + LenRead;

        //             ReadRecord_(request     :=  StartRW,
        //                         id          :=  Inputs.HardwareId,
        //                         index       :=  16#b02e,
        //                         maxLength   :=  _lenght,
        //                         record      :=  RD_Data,
        //                         status      =>  RD_Status,
        //                         length      =>  LengthRead);

        //             IF ReadRecord_.VALID AND NOT ReadRecord_.BUSY THEN
        //                 ErrorCounter := UINT#0;
        //                 State := 55;
        //             ELSIF ReadRecord_.ERROR THEN
        //                 tmpWord := TO_WORD(TO_DINT(RD_Status)/256);
        //                 wordhlp := tmpWord;
        //                 //try it again
        //                 IF ((tmpWord = WORD#16#80A7) OR (tmpWord = WORD#16#80B5) OR (tmpWord = WORD#16#80C0) OR (tmpWord = WORD#16#80C1) OR (tmpWord = WORD#16#80C2)
        //                     OR (tmpWord = WORD#16#80C3) OR (tmpWord = WORD#16#80C4)) AND (ErrorCounter < MaxRetryCounter) THEN
        //                     ErrorCounter := ErrorCounter + UINT#1;
        //                     StartRW := false;
        //                     StartTimer := TRUE;
        //                 ELSE
        //                     State := 80;
        //                 END_IF;
        //             END_IF;
        //         END_IF;

        //         IF State = 55 THEN //Reading finished
        //             CASE TO_INT(RD_Data[4]) OF // Format
        //                 0:  //reserved
        //                     Outputs.ValueReadREAL := 0;
        //                     Outputs.ValueReadLINT := 0;
        //                     Outputs.ValueReadBOOL := FALSE;

        //                     Outputs.ErrorId := DWORD#16#1001;    //reserved DataType
        //                     // #Error
        //                     State := 200;

        //                 1, 2, 3, 4, 5, 6, 7, 8, 55, 56, 65, 66, 67:
        //                     State := 60;

        //                 68:  //Error
        //                     tmpDWord.%B0 := RD_Data[7];
        //                     tmpDWord.%B1 := RD_Data[6];
        //                     Outputs.ErrorId := tmpDWord OR PD_Error;

        //                     //copy the value to the output
        //                     Outputs.ValueReadREAL := 0;
        //                     Outputs.ValueReadLINT := 0;
        //                     Outputs.ValueReadBOOL := FALSE;

        //                     // #Error
        //                     State := 200;

        //                 ELSE
        //                     Outputs.ValueReadREAL := 0;
        //                     Outputs.ValueReadLINT := 0;
        //                     Outputs.ValueReadBOOL := FALSE;

        //                     Outputs.ErrorId := DWORD#16#1000;    //unknown DataType
        //                     // #Error
        //                     State := 200;
        //             END_CASE;
        //         END_IF;

        //         IF State = 60 THEN //reading Done from Write request
        //             (* ------------------ HEADER --------------------*)
        //             //Request reference starts with 1 and will count up
        //             WR_Data[0] := TO_BYTE(TO_INT(ReqRef) + 1);
        //             // Requst ID = 2 (Change Parameter)
        //             WR_Data[1] := BYTE#2;
        //             //Fill the Axis number
        //             WR_Data[2] := Inputs.AxisNo;
        //             // Single parameter access
        //             WR_Data[3] := BYTE#1;
        //             (* ------------------ DATA --------------------*)
        //             // Attribute
        //             WR_Data[4] := BYTE#16#10;
        //             // Single Access
        //             WR_Data[5] := BYTE#1;
        //             // PNU
        //             WR_Data[6] := Inputs.ParameterNo.%B1;
        //             WR_Data[7] := Inputs.ParameterNo.%B0;
        //             // Subindex
        //             WR_Data[8] := Inputs.Subindex.%B1;
        //             WR_Data[9] := Inputs.Subindex.%B0;
        //             //Format
        //             WR_Data[10] := RD_Data[4];
        //             //No. Values
        //             WR_Data[11] := BYTE#1;
        //             //erase send buffer
        //             FOR i := 12 TO 19 DO
        //                 WR_Data[i] := BYTE#0;
        //             END_FOR;

        //             CASE TO_INT(RD_Data[4]) OF //Format
        //                 0:  //reserved
        //                     Outputs.ValueReadREAL := 0;
        //                     Outputs.ValueReadLINT := 0;
        //                     Outputs.ValueReadBOOL := FALSE;

        //                     Outputs.ErrorId := DWORD#16#1001;    //reserved DataType
        //                     // #Error
        //                     State := 200;

        //                 1:  //BOOL
        //                     WR_Data[12] := TO_BYTE(Inputs.ValueWriteBOOL);

        //                 2, 5, 65:  //SINT8, USINT8, BYTE
        //                     WR_Data[12] := TO_BYTE(Inputs.ValueWriteLINT);

        //                 3, 6, 66:  //SINT16, UINT16, WORD
        //                     WR_Data[12] := Inputs.ValueWriteLINT.%B1;
        //                     WR_Data[13] := Inputs.ValueWriteLINT.%B0;

        //                 4, 7, 67: //SINT32, UDINT32, DWORD
        //                     WR_Data[12] := Inputs.ValueWriteLINT.%B3;
        //                     WR_Data[13] := Inputs.ValueWriteLINT.%B2;
        //                     WR_Data[14] := Inputs.ValueWriteLINT.%B1;
        //                     WR_Data[15] := Inputs.ValueWriteLINT.%B0;

        //                 8:  //FLOAT32
        //                     tmpDWORD    :=  TO_DWORD(Inputs.ValueWriteREAL);
        //                     WR_Data[12] := tmpDWORD.%B3;
        //                     WR_Data[13] := tmpDWORD.%B2;
        //                     WR_Data[14] := tmpDWORD.%B1;
        //                     WR_Data[15] := tmpDWORD.%B0;

        //                 55, 56:  //SINT64
        //                     WR_Data[12] := Inputs.ValueWriteLINT.%B7;
        //                     WR_Data[13] := Inputs.ValueWriteLINT.%B6;
        //                     WR_Data[14] := Inputs.ValueWriteLINT.%B5;
        //                     WR_Data[15] := Inputs.ValueWriteLINT.%B4;
        //                     WR_Data[16] := Inputs.ValueWriteLINT.%B3;
        //                     WR_Data[17] := Inputs.ValueWriteLINT.%B2;
        //                     WR_Data[18] := Inputs.ValueWriteLINT.%B1;
        //                     WR_Data[19] := Inputs.ValueWriteLINT.%B0;

        //             END_CASE;

        //             //goto the next step
        //             State := 61;
        //         END_IF;

        //         IF State = 61 THEN //send the write Request
        //             // Lenght of the telegramm to be send
        //             _lenght := LenHeader + LenWrite;

        //             WriteRecord_(request    :=  StartRW,
        //                         id          :=  Inputs.HardwareId,
        //                         index       :=  16#b02e,
        //                         length      :=  _lenght,
        //                         record      :=  WR_Data,
        //                         status      =>  RW_Status);

        //             IF WriteRecord_.DONE THEN
        //                 State := 62;
        //             ELSIF WriteRecord_.ERROR THEN
        //                 tmpWord := TO_WORD(TO_DINT(RW_Status)/256);
        //                 wordhlp := tmpWord;
        //                 //try it again
        //                 IF ((tmpWord = WORD#16#80A7) OR (tmpWord = WORD#16#80B5) OR (tmpWord = WORD#16#80C0) OR (tmpWord = WORD#16#80C1) OR (tmpWord = WORD#16#80C2)
        //                     OR (tmpWord = WORD#16#80C3) OR (tmpWord = WORD#16#80C4)) AND (ErrorCounter < MaxRetryCounter) THEN
        //                     ErrorCounter := ErrorCounter + UINT#1;
        //                     StartRW := FALSE;
        //                     StartTimer := TRUE;
        //                 ELSE
        //                     State := 90;
        //                 END_IF;
        //             END_IF;
        //         END_IF;

        //         IF State = 62 THEN //Read the answer of the write request

        //             //delete old response values
        //             FOR i := 0 TO 13 DO
        //                 RD_Data[i] := BYTE#0;
        //             END_FOR;

        //             // Lenght of the telegramm for reading
        //             _lenght := LenHeader + LenRead;

        //             ReadRecord_(request     :=  StartRW,
        //                         id          :=  Inputs.HardwareId,
        //                         index       :=  16#b02e,
        //                         maxLength   :=  _lenght,
        //                         record      :=  RD_Data,
        //                         status      =>  RD_Status,
        //                         length      =>  LengthRead);

        //             IF ReadRecord_.VALID AND NOT ReadRecord_.BUSY THEN
        //                 ErrorCounter := UINT#0;
        //                 State := 63;
        //             ELSIF ReadRecord_.ERROR THEN
        //                 tmpWord := TO_WORD(TO_DINT(RD_Status)/256);
        //                 wordhlp := tmpWord;
        //                 //try it again
        //                 IF ((tmpWord = WORD#16#80A7) OR (tmpWord = WORD#16#80B5) OR (tmpWord = WORD#16#80C0) OR (tmpWord = WORD#16#80C1) OR (tmpWord = WORD#16#80C2)
        //                     OR (tmpWord = WORD#16#80C3) OR (tmpWord = WORD#16#80C4)) AND (ErrorCounter < MaxRetryCounter) THEN
        //                     ErrorCounter := ErrorCounter + UINT#1;
        //                     StartRW := FALSE;
        //                     StartTimer := TRUE;
        //                 ELSE
        //                     State := 80;
        //                 END_IF;
        //             END_IF;
        //         END_IF;

        //         IF State = 63 THEN //Reading finished

        //             CASE TO_INT(RD_Data[1]) OF //ReqId

        //                 2:  //positive resonse
        //                     State := 150;

        //                 128..130:  //negative response
        //                     IF RD_Data[4] = BYTE#68 THEN //Format
        //                         tmpDWord.%B0 := RD_Data[7];
        //                         tmpDWord.%B1 := RD_Data[6];
        //                         Outputs.ErrorId := tmpDWord OR PD_Error;

        //                         // #Error
        //                         State := 200;
        //                     ELSE
        //                         Outputs.ErrorId := DWORD#16#1003; //negative response without error code
        //                         State := 300;
        //                     END_IF;
        //                 ELSE  //undefined response ID
        //                     Outputs.ErrorId := DWORD#16#1002;
        //                     State := 300;
        //             END_CASE;
        //         END_IF;

        //         IF State = 70 THEN // Error while ReadWrite Access
        //             Outputs.Done := TRUE;
        //             Outputs.Busy := FALSE;
        //             Outputs.Error := TRUE;
        //             Outputs.ErrorId := WR_Status;
        //         END_IF;

        //         IF State = 80 THEN //Error Reading Access
        //             Outputs.Done := TRUE;
        //             Outputs.Busy := FALSE;
        //             Outputs.Error := TRUE;
        //             Outputs.ErrorId := RD_Status;
        //         END_IF;

        //         IF State = 90 THEN // Error while Write Access
        //             Outputs.Done := TRUE;
        //             Outputs.Busy := FALSE;
        //             Outputs.Error := TRUE;
        //             Outputs.ErrorId := RW_Status;
        //         END_IF;

        //         IF State = 100 THEN // read successfully
        //             Outputs.Done := TRUE;
        //             Outputs.Busy := FALSE;
        //             Outputs.Error := FALSE;
        //         END_IF;

        //         IF State = 150 THEN // write successfully
        //             Outputs.Done := TRUE;
        //             Outputs.Busy := FALSE;
        //             Outputs.Error := FALSE;
        //         END_IF;

        //         IF State = 200 THEN //Error while reading
        //             Outputs.Done := TRUE;
        //             Outputs.Busy := FALSE;
        //             Outputs.Error := TRUE;

        //             IF State = 300 THEN //Error while writing
        //                 Outputs.Done := TRUE;
        //                 Outputs.Busy := FALSE;
        //                 Outputs.Error := TRUE;
        //             END_IF;
        //         END_IF;

        //         IF NOT Inputs.Enable THEN
        //             State := 0;
        //             ReqRef := BYTE#1;
        //             Outputs.Done := FALSE;
        //             Outputs.Busy := FALSE;
        //             Outputs.Error := FALSE;
        //             Outputs.ErrorId := DWORD#16#00000000;
        //             Outputs.ValueReadBOOL := FALSE;
        //             Outputs.ValueReadLINT := 0;
        //             Outputs.ValueReadREAL := 0;
        //             RD_Status := DWORD#0;
        //             ErrorCounter := UINT#0;
        //         END_IF;

        //         Enable_PV := Inputs.Enable;

        // END_METHOD

        METHOD PUBLIC Restore
            VAR
                i : INT;
            END_VAR

            State := 0;
            ReqRef := BYTE#1;
            Outputs.Done := FALSE;
            Outputs.Busy := FALSE;
            Outputs.Error := FALSE;
            Outputs.ErrorId := DWORD#16#00000000;
            Outputs.ValueReadBOOL := FALSE;
            Outputs.ValueReadLINT := 0;
            Outputs.ValueReadREAL := 0;
            RD_Status := DWORD#0;
            ErrorCounter := UINT#0;
            Enable_PV      := FALSE;
            Busy_	:= FALSE;
            Done_	:= FALSE;
            Error_	:= FALSE;
            ErrorId_:= FALSE;
            StartTimer := FALSE;
            StartRW := FALSE;

            AxoOnDelatTimer.OnDelay(THIS, FALSE,T#0MS);
            FOR i := 0 TO 9 DO
                RW_Data[i] := BYTE#0;
            END_FOR;
            FOR i := 0 TO 19 DO
                WR_Data[i] := BYTE#0;
            END_FOR;
            FOR i := 0 TO 13 DO
                RD_Data[i] := BYTE#0;
            END_FOR;

            RW_Status        :=	DWORD#0;
            WR_Status        :=	DWORD#0;
            RD_Status        :=	DWORD#0;

            ReadRecord_(request    :=  FALSE, record      :=  RW_Data);
            WriteRecord_(request    :=  FALSE, record      :=  RW_Data);
            ErrorCounter    :=	UINT#0;

            LengthRead      :=	UINT#0;
            wordhlp         :=   WORD#0;
        END_METHOD
    END_CLASS
END_NAMESPACE

(* ---- PROFIdriveTelegram_111.st ---- *)
NAMESPACE AXOpen.Components.Festo.Drives

    {#ix-attr:[Container(Layout.Stack)]}
    {S7.extern=ReadWrite}
    CLASS PUBLIC PROFIdriveTelegram_111_STW1
        VAR PUBLIC
            {#ix-attr:[Container(Layout.Stack)]}
            {#ix-set:AttributeName = "<#jog1#>"}
            jog1    :  BOOL;
            {#ix-set:AttributeName = "<#jog2#>"}
            jog2    :  BOOL;
            {#ix-set:AttributeName = "<#controlByPlc#>"}
            controlByPlc    :  BOOL;
            {#ix-set:AttributeName = "<#StartHoming#>"}
            StartHoming :  BOOL;
            {#ix-set:AttributeName = "<#ReleaseBrake#>"}
            ReleaseBrake    :  BOOL;
            {#ix-set:AttributeName = "<#ExternalBlockChange#>"}
            ExternalBlockChange :  BOOL;
            {#ix-set:AttributeName = "<#reserved14#>"}
            reserved14  :  BOOL;
            {#ix-set:AttributeName = "<#reserved15#>"}
            reserved15  :  BOOL;
            {#ix-set:AttributeName = "<#on#>"}
            on_  :  BOOL;
            {#ix-set:AttributeName = "<#noCoastStop#>"}
            noCoastStop :  BOOL;
            {#ix-set:AttributeName = "<#noQuickStop#>"}
            noQuickStop :  BOOL;
            {#ix-set:AttributeName = "<#enableOperation#>"}
            enableOperation :  BOOL;
            {#ix-set:AttributeName = "<#cancelTraversing#>"}
            cancelTraversing    :  BOOL;
            {#ix-set:AttributeName = "<#intermediateStop#>"}
            intermediateStop    :  BOOL;
            {#ix-set:AttributeName = "<#activateTraversing#>"}
            activateTraversing  :  BOOL;
            {#ix-set:AttributeName = "<#acknowledgeFault#>"}
            acknowledgeFault    :  BOOL;
        END_VAR
    END_CLASS

    {#ix-attr:[Container(Layout.Stack)]}
    {S7.extern=ReadWrite}
    CLASS PUBLIC PROFIdriveTelegram_111_POS_STW1
        VAR PUBLIC
            {#ix-attr:[Container(Layout.Stack)]}
            {#ix-set:AttributeName = "<#MDI_MOD#>"}
            MDI_MOD    :  BOOL;
            {#ix-set:AttributeName = "<#PosModulo#>"}
            PosModulo    :  BOOL;
            {#ix-set:AttributeName = "<#NegModulo#>"}
            NegModulo    :  BOOL;
            {#ix-set:AttributeName = "<#reserved11#>"}
            reserved11 :  BOOL;
            {#ix-set:AttributeName = "<#reserved12#>"}
            reserved12    :  BOOL;
            {#ix-set:AttributeName = "<#reserved13#>"}
            reserved13 :  BOOL;
            {#ix-set:AttributeName = "<#SetupMode#>"}
            SetupMode  :  BOOL;
            {#ix-set:AttributeName = "<#MDI_Activate#>"}
            MDI_Activate  :  BOOL;
            {#ix-set:AttributeName = "<#travBlockBit0#>"}
            travBlockBit0  :  BOOL;
            {#ix-set:AttributeName = "<#travBlockBit1#>"}
            travBlockBit1 :  BOOL;
            {#ix-set:AttributeName = "<#travBlockBit2#>"}
            travBlockBit2 :  BOOL;
            {#ix-set:AttributeName = "<#travBlockBit3#>"}
            travBlockBit3 :  BOOL;
            {#ix-set:AttributeName = "<#travBlockBit4#>"}
            travBlockBit4    :  BOOL;
            {#ix-set:AttributeName = "<#travBlockBit5#>"}
            travBlockBit5  :  BOOL;
            {#ix-set:AttributeName = "<#travBlockBit6#>"}
            travBlockBit6    :  BOOL;
            {#ix-set:AttributeName = "<#reserved7#>"}
            reserved7    :  BOOL;
        END_VAR
    END_CLASS

    {#ix-attr:[Container(Layout.Stack)]}
    {S7.extern=ReadWrite}
    CLASS PUBLIC PROFIdriveTelegram_111_POS_STW2
        VAR PUBLIC
            {#ix-attr:[Container(Layout.Stack)]}
            {#ix-set:AttributeName = "<#FlyingRef#>"}
            FlyingRef    :  BOOL;
            {#ix-set:AttributeName = "<#reserved9#>"}
            reserved9    :  BOOL;
            {#ix-set:AttributeName = "<#SelectProbe#>"}
            SelectProbe    :  BOOL;
            {#ix-set:AttributeName = "<#ProbeEdgeEval#>"}
            ProbeEdgeEval :  BOOL;
            {#ix-set:AttributeName = "<#reserved12#>"}
            reserved12    :  BOOL;
            {#ix-set:AttributeName = "<#reserved13#>"}
            reserved13 :  BOOL;
            {#ix-set:AttributeName = "<#SW-Limit#>"}
            SW_Limit  :  BOOL;
            {#ix-set:AttributeName = "<#HW-Limit#>"}
            HW_Limit  :  BOOL;
            {#ix-set:AttributeName = "<#Trackingmode#>"}
            Trackingmode  :  BOOL;
            {#ix-set:AttributeName = "<#SetReferencePoint#>"}
            SetReferencePoint :  BOOL;
            {#ix-set:AttributeName = "<#reserved2#>"}
            reserved2 :  BOOL;
            {#ix-set:AttributeName = "<#reserved3#>"}
            reserved3 :  BOOL;
            {#ix-set:AttributeName = "<#reserved4#>"}
            reserved4    :  BOOL;
            {#ix-set:AttributeName = "<#jog_inc#>"}
            jog_inc  :  BOOL;
            {#ix-set:AttributeName = "<#reserved6#>"}
            reserved6    :  BOOL;
            {#ix-set:AttributeName = "<#reserved7#>"}
            reserved7    :  BOOL;
        END_VAR
    END_CLASS

    {#ix-attr:[Container(Layout.Stack)]}
    {S7.extern=ReadWrite}
    CLASS PUBLIC PROFIdriveTelegram_111_STW2
        VAR PUBLIC
            {#ix-attr:[Container(Layout.Stack)]}
            {#ix-set:AttributeName = "<#TravelToFixStop#>"}
            TravelToFixStop    :  BOOL;
            {#ix-set:AttributeName = "<#reserved9#>"}
            reserved9    :  BOOL;
            {#ix-set:AttributeName = "<#reserved10#>"}
            reserved10    :  BOOL;
            {#ix-set:AttributeName = "<#reserved11#>"}
            reserved11 :  BOOL;
            {#ix-set:AttributeName = "<#signOfLifeBit0#>"}
            signOfLifeBit0    :  BOOL;
            {#ix-set:AttributeName = "<#signOfLifeBit1#>"}
            signOfLifeBit1 :  BOOL;
            {#ix-set:AttributeName = "<#signOfLifeBit2#>"}
            signOfLifeBit2  :  BOOL;
            {#ix-set:AttributeName = "<#signOfLifeBit3#>"}
            signOfLifeBit3  :  BOOL;
            {#ix-set:AttributeName = "<#reserved0#>"}
            reserved0  :  BOOL;
            {#ix-set:AttributeName = "<#reserved1#>"}
            reserved1 :  BOOL;
            {#ix-set:AttributeName = "<#reserved2#>"}
            reserved2 :  BOOL;
            {#ix-set:AttributeName = "<#reserved3#>"}
            reserved3 :  BOOL;
            {#ix-set:AttributeName = "<#reserved4#>"}
            reserved4    :  BOOL;
            {#ix-set:AttributeName = "<#reserved5#>"}
            reserved5    :  BOOL;
            {#ix-set:AttributeName = "<#reserved6#>"}
            reserved6  :  BOOL;
            {#ix-set:AttributeName = "<#reserved7#>"}
            reserved7    :  BOOL;
        END_VAR
    END_CLASS

    {#ix-attr:[Container(Layout.Wrap)]}
    {S7.extern=ReadWrite}
    CLASS PUBLIC PROFIdriveTelegram_111_OUT
        VAR PUBLIC
            {#ix-attr:[Container(Layout.Wrap)]}
            {#ix-attr:[Group(GroupLayout.GroupBox)]}
            {#ix-set:AttributeName = "<#STW1#>"}
            STW1      :   PROFIdriveTelegram_111_STW1;
            {#ix-attr:[Container(Layout.Wrap)]}
            {#ix-attr:[Group(GroupLayout.GroupBox)]}
            {#ix-set:AttributeName = "<#POS_STW1#>"}
            POS_STW1      :   PROFIdriveTelegram_111_POS_STW1;
            {#ix-attr:[Container(Layout.Wrap)]}
            {#ix-attr:[Group(GroupLayout.GroupBox)]}
            {#ix-set:AttributeName = "<#POS_STW2#>"}
            POS_STW2      :   PROFIdriveTelegram_111_POS_STW2;
            {#ix-attr:[Container(Layout.Wrap)]}
            {#ix-attr:[Group(GroupLayout.GroupBox)]}
            {#ix-set:AttributeName = "<#STW2#>"}
            STW2      :   PROFIdriveTelegram_111_STW2;
            {#ix-attr:[Container(Layout.Stack)]}
            {#ix-set:AttributeName = "<#Override#>"}
            Override_    :	WORD;
            {#ix-set:AttributeName = "<#MDI_TARPOS#>"}
            MDI_TARPOS  :	DINT;
            {#ix-set:AttributeName = "<#MDI_VELOCITY#>"}
            MDI_VELOCITY    :	DINT;
            {#ix-set:AttributeName = "<#MDI_ACC#>"}
            MDI_ACC :	UINT;
            {#ix-set:AttributeName = "<#MDI_DEC#>"}
            MDI_DEC :	UINT;
            {#ix-set:AttributeName = "<#reserved11#>"}
            reserved11  :	WORD;

        END_VAR
    END_CLASS

    {#ix-attr:[Container(Layout.Stack)]}
    {S7.extern=ReadWrite}
    CLASS PUBLIC PROFIdriveTelegram_111_ZSW1
        VAR PUBLIC
            {#ix-attr:[Container(Layout.Stack)]}
            {#ix-set:AttributeName = "<#followingErrorInTolerance#> (X8)"}
            followingErrorInTolerance    :  BOOL;
            {#ix-set:AttributeName = "<#controlRequest#> (X9)"}
            controlRequest    :  BOOL;
            {#ix-set:AttributeName = "<#targetPosReached#> (X10)"}
            targetPosReached    :  BOOL;
            {#ix-set:AttributeName = "<#homePosSet#> (X11)"}
            homePosSet :  BOOL;
            {#ix-set:AttributeName = "<#acknowledgeTraversingBlockActivated#> (X12)"}
            acknowledgeTraversingBlockActivated    :  BOOL;
            {#ix-set:AttributeName = "<#driveStopped#> (X13)"}
            driveStopped :  BOOL;
            {#ix-set:AttributeName = "<#axisAccelerates#> (X14)"}
            axisAccelerates  :  BOOL;
            {#ix-set:AttributeName = "<#axisDecelerates#> (X15)"}
            axisDecelerates  :  BOOL;
            {#ix-set:AttributeName = "<#readyForSwitchOn#> (X0)"}
            readyForSwitchOn  :  BOOL;
            {#ix-set:AttributeName = "<#ready#> (X1)"}
            ready :  BOOL;
            {#ix-set:AttributeName = "<#operationEnabled#> (X2)"}
            operationEnabled :  BOOL;
            {#ix-set:AttributeName = "<#faultPresent#> (X3)"}
            faultPresent :  BOOL;
            {#ix-set:AttributeName = "<#noCoastingActive#> (X4)"}
            noCoastingActive    :  BOOL;
            {#ix-set:AttributeName = "<#noQuickStopActive#> (X5)"}
            noQuickStopActive    :  BOOL;
            {#ix-set:AttributeName = "<#switchingOnInhibitedActive#> (X6)"}
            switchingOnInhibitedActive  :  BOOL;
            {#ix-set:AttributeName = "<#warningActive#> (X7)"}
            warningActive    :  BOOL;
        END_VAR
    END_CLASS

    {#ix-attr:[Container(Layout.Stack)]}
    {S7.extern=ReadWrite}
    CLASS PUBLIC PROFIdriveTelegram_111_ZSW2
        VAR PUBLIC
            {#ix-attr:[Container(Layout.Stack)]}
            {#ix-set:AttributeName = "<#deviceSpecificBit8#>"}
            deviceSpecificBit8    :  BOOL;
            {#ix-set:AttributeName = "<#deviceSpecificBit9#>"}
            deviceSpecificBit9    :  BOOL;
            {#ix-set:AttributeName = "<#deviceSpecificBit10#>"}
            deviceSpecificBit10    :  BOOL;
            {#ix-set:AttributeName = "<#deviceSpecificBit11#>"}
            deviceSpecificBit11 :  BOOL;
            {#ix-set:AttributeName = "<#doSignOfLifeBit0#>"}
            doSignOfLifeBit0    :  BOOL;
            {#ix-set:AttributeName = "<#doSignOfLifeBit1#>"}
            doSignOfLifeBit1 :  BOOL;
            {#ix-set:AttributeName = "<#doSignOfLifeBit2#>"}
            doSignOfLifeBit2  :  BOOL;
            {#ix-set:AttributeName = "<#doSignOfLifeBit3#>"}
            doSignOfLifeBit3  :  BOOL;
            {#ix-set:AttributeName = "<#deviceSpecificBit0#>"}
            deviceSpecificBit0  :  BOOL;
            {#ix-set:AttributeName = "<#deviceSpecificBit1#>"}
            deviceSpecificBit1 :  BOOL;
            {#ix-set:AttributeName = "<#deviceSpecificBit2#>"}
            deviceSpecificBit2 :  BOOL;
            {#ix-set:AttributeName = "<#deviceSpecificBit3#>"}
            deviceSpecificBit3 :  BOOL;
            {#ix-set:AttributeName = "<#deviceSpecificBit4#>"}
            deviceSpecificBit4    :  BOOL;
            {#ix-set:AttributeName = "<#deviceSpecificBit5#>"}
            deviceSpecificBit5    :  BOOL;
            {#ix-set:AttributeName = "<#deviceSpecificBit6#>"}
            deviceSpecificBit6  :  BOOL;
            {#ix-set:AttributeName = "<#deviceSpecificBit7#>"}
            deviceSpecificBit7    :  BOOL;
        END_VAR
    END_CLASS

    {#ix-attr:[Container(Layout.Wrap)]}
    {S7.extern=ReadWrite}
    CLASS PUBLIC PROFIdriveTelegram_111_IN
        VAR PUBLIC
            {#ix-attr:[Container(Layout.Wrap)]}
            {#ix-attr:[Group(GroupLayout.GroupBox)]}
            {#ix-set:AttributeName = "<#ZSW1#>"}
            ZSW1      :   PROFIdriveTelegram_111_ZSW1;
            {#ix-attr:[Container(Layout.Stack)]}
            {#ix-set:AttributeName = "<#POS_ZSW1#>"}
            POS_ZSW1      :   WORD;
            {#ix-set:AttributeName = "<#POS_ZSW2#>"}
            POS_ZSW2      :   WORD;
            {#ix-attr:[Container(Layout.Stack)]}
            {#ix-attr:[Group(GroupLayout.GroupBox)]}
            {#ix-set:AttributeName = "<#ZSW2#>"}
            ZSW2      :   PROFIdriveTelegram_111_ZSW2;
            {#ix-attr:[Container(Layout.Stack)]}
            {#ix-set:AttributeName = "<#MELDW#>"}
            MELDW    :	WORD;
            {#ix-set:AttributeName = "<#XIST_A#>"}
            XIST_A  :	DINT;
            {#ix-set:AttributeName = "<#NIST_B#>"}
            NIST_B    :	DINT;
            {#ix-set:AttributeName = "<#Fault_Code#>"}
            Fault_Code :	UINT;
            {#ix-set:AttributeName = "<#Warn_Code#>"}
            Warn_Code :	UINT;
            {#ix-set:AttributeName = "<#Reserved#>"}
            Reserved  :	WORD;
        END_VAR
    END_CLASS

    {#ix-attr:[Container(Layout.Wrap)]}
    {S7.extern=ReadWrite}
    CLASS PUBLIC PROFIdriveTelegram_111
        VAR PUBLIC
            {#ix-attr:[Container(Layout.Wrap)]}
            {#ix-attr:[Group(GroupLayout.GroupBox)]}
            {#ix-set:AttributeName = "<#OUT#>"}
            OUT      :   PROFIdriveTelegram_111_OUT;
            {#ix-attr:[Container(Layout.Wrap)]}
            {#ix-attr:[Group(GroupLayout.GroupBox)]}
            {#ix-set:AttributeName = "<#IN#>"}
            IN      :   PROFIdriveTelegram_111_IN;
        END_VAR
    END_CLASS
END_NAMESPACE

(* ---- PROFIdriveTelegram_750.st ---- *)
NAMESPACE AXOpen.Components.Festo.Drives

    {#ix-attr:[Container(Layout.Wrap)]}
    {S7.extern=ReadWrite}
    CLASS PUBLIC PROFIdriveTelegram_750_OUT
        VAR PUBLIC
            {#ix-attr:[Container(Layout.Stack)]}
            {#ix-set:AttributeName = "<#M_ADD1#>"}
            M_ADD1    :	INT;
            {#ix-set:AttributeName = "<#M_LIMIT_POS#>"}
            M_LIMIT_POS  :	INT;
            {#ix-set:AttributeName = "<#M_LIMIT_NEG#>"}
            M_LIMIT_NEG    :	INT;
            {#ix-set:AttributeName = "<#Reserved#>"}
            Reserved :	WORD;
        END_VAR
    END_CLASS

    {#ix-attr:[Container(Layout.Wrap)]}
    {S7.extern=ReadWrite}
    CLASS PUBLIC PROFIdriveTelegram_750_IN
        VAR PUBLIC
            {#ix-attr:[Container(Layout.Stack)]}
            {#ix-set:AttributeName = "<#M_Actual#>"}
            M_Actual    :	INT;
        END_VAR
    END_CLASS

    {#ix-attr:[Container(Layout.Wrap)]}
    {S7.extern=ReadWrite}
    CLASS PUBLIC PROFIdriveTelegram_750
        VAR PUBLIC
            {#ix-attr:[Container(Layout.Wrap)]}
            {#ix-attr:[Group(GroupLayout.GroupBox)]}
            {#ix-set:AttributeName = "<#OUT#>"}
            OUT      :   PROFIdriveTelegram_750_OUT;
            {#ix-attr:[Container(Layout.Wrap)]}
            {#ix-attr:[Group(GroupLayout.GroupBox)]}
            {#ix-set:AttributeName = "<#IN#>"}
            IN      :   PROFIdriveTelegram_750_IN;
        END_VAR
    END_CLASS
END_NAMESPACE
